{attribute 'GeneratedUsingTerminal: EL3314-0002-0016'}
{attribute addProperty BoxType "EL3314-0002-0016"}
{attribute addProperty Id "StatusAT %I*Status_F2CE6D917ValueAT %I*DINT4"}
{attribute addProperty CRC "1159803140"}
{attribute addProperty Size "11"}
TYPE TC_Inputs_Channel_45213104 :
STRUCT
	{attribute addProperty Name "Status"}
	Status AT %I* : Status_F2CE6D91;
	{attribute addProperty Name "Value"}
	Value AT %I* : DINT;
END_STRUCT
END_TYPE

(* stored: Version 1.2.0.0, ProductVersion 3.1.4024.9
   DUT TC_Inputs_Channel_45213104: Id {af0fe86c-e8aa-4561-bc23-be484350b610} *)
